TYPE "UDT_UDPFrame"
VERSION : 0.1
   STRUCT
      "type" : String;
      index : Int;
      data : Array[0..511] of Byte;
      remote_ip : USInt;
   END_STRUCT;

END_TYPE

